// TIA Portal V16 export
// export: Created 2022-09-01T13:37:26.7325427Z, ExportSetting WithDefaults, DisplayName Totally Integrated Automation Portal, DisplayVersion V16, DisplayName TIA Portal Version Control Interface, DisplayVersion V16, DisplayName TIA Portal Openness, DisplayVersion V16, DisplayName STEP 7 Professional, DisplayVersion V16, DisplayName STEP 7 Safety, DisplayVersion V16, DisplayName WinCC Advanced, DisplayVersion V16
VAR_GLOBAL   // PLC tag table "Analógicas"
   FQ301_MEDIDOR_CAUDAL AT %IW16 : Word;
   PC401_SENSOR_PRESSÃO AT %IW18 : Word;
END_VAR
